(* CoDeSys 2.3 export: E_FROELINGANLAGENZUSTAND.EXP *)

(* Data type *)
TYPE E_FroelingAnlagenzustand : (
	Winterbetrieb := 0,
	Sommerbetrieb := 1,
	Uebergangsbetrieb := 2,
	KeinScheitholzbetrieb := 3,
	Ausgeschaltet := 5,
	Extraheizen := 6,
	Kaminkehrer := 7,
	Reinigen := 8
);
END_TYPE
